{attribute 'pack_mode' := '2'}
TYPE stEL3318_Channel:
STRUCT
	Status 	AT %I* : stEL3318_ChannelStatus;	 
	Value 	AT %I* : WORD;  
END_STRUCT
END_TYPE;

(* stored: Version 1.1.0.1, ProductVersion 3.1.4024.4
   DUT stEL3318_Channel: Id {9e196651-bc71-4a31-936a-8265a94162e2} *)
